FUNCTION_BLOCK L0_8070Service (* FAGOR 8070 CNC service FB *)
  (* Standard: 61499-2; Description: This FB is the entry point of the CNC service *)
  (* Version 0.0, 2014-09-01, EQUEROL, UJI *)
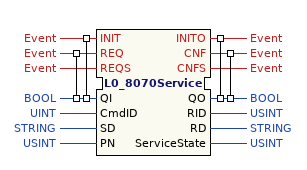
  EVENT_INPUT
    INIT WITH QI; (* Initialization Request *)
    REQ WITH QI; (* Normal Execution Request *)
    REQS; (* Request Service state *)
  END_EVENT
  EVENT_OUTPUT
    INITO WITH QO; (* Initialization Confirm *)
    CNF WITH QO; (* Execution Confirmation *)
    CNFS; (* Service State Confirmation *)
  END_EVENT
  VAR_INPUT
    QI : BOOL; (* Input event qualifier *)
    CmdID : UINT; (* Action to be executed ID *)
    SD : STRING; (* Action parameters *)
    PN : USINT; (* Number of parameters *)
  END_VAR
  VAR_OUTPUT
    QO : BOOL; (* Output event qualifier *)
    RID : USINT; (* Executed action ID *)
    RD : STRING; (* Service feedback data *)
    ServiceState : USINT; (* CNC Service state *)
  END_VAR
  FBS
    L0_State : L0_State;
    L0_SendBlk : L0_SendBlk;
    L0_CNCEncap : L0_CNCEncap;
    L0_IncomEx : L0_IncomEx;
    L0_StateHandler : L0_StateHandler;
    L0_CompletedEx : L0_CompletedEx;
    CM_Merge2E2USINT : CM_Merge2E2USINT;
    CM_Merge2E2USINT_0 : CM_Merge2E2USINT(E1In := 3, E2In := 4);
    CM_ChkService : CM_ChkService;
    CM_Merge2E2USINT_1 : CM_Merge2E2USINT;
    L0_ReqManager : L0_ReqManager;
    L0_InitService : L0_InitService;
  END_FBS
  EVENT_CONNECTIONS
    L0_SendBlk.IND TO L0_State.UPDT;
    L0_CNCEncap.CNF TO L0_SendBlk.REQ;
    L0_CNCEncap.INITO TO L0_SendBlk.INIT;
    L0_SendBlk.INITO TO L0_State.INIT;
    L0_StateHandler.OnInterrupted TO L0_IncomEx.Interrupted;
    L0_StateHandler.OnIntError TO L0_IncomEx.InterrupErr;
    L0_StateHandler.OnReady TO L0_CompletedEx.OnReady;
    L0_StateHandler.OnExecution TO L0_CompletedEx.OnExecuting;
    L0_StateHandler.OnNotReady TO L0_CompletedEx.OnNotReady;
    L0_CompletedEx.Success TO CM_Merge2E2USINT.E1;
    L0_IncomEx.CNF TO CM_Merge2E2USINT.E2;
    L0_State.UPDTO TO L0_StateHandler.REQ;
    CM_ChkService.BUSY TO CM_Merge2E2USINT_0.E2;
    CM_ChkService.DOWN TO CM_Merge2E2USINT_0.E1;
    CM_ChkService.UP TO L0_ReqManager.REQ;
    CM_ChkService.REQS TO L0_State.REQ;
    CM_Merge2E2USINT_0.EO TO CM_Merge2E2USINT_1.E2;
    L0_ReqManager.IND TO CM_Merge2E2USINT_1.E1;
    CM_Merge2E2USINT.EO TO L0_ReqManager.UPDT;
    CM_Merge2E2USINT_1.EO TO CNF;
    REQS TO L0_State.REQ;
    L0_State.CNF TO CNFS;
    L0_State.CNF TO CM_ChkService.RSP;
    REQ TO CM_ChkService.REQ;
    INIT TO L0_InitService.INIT;
    L0_InitService.INITOSer TO L0_ReqManager.INIT;
    L0_ReqManager.INITO TO L0_CNCEncap.INIT;
    L0_State.INITO TO L0_InitService.INITSer;
    L0_InitService.INITO TO INITO;
  END_CONNECTIONS
  DATA_CONNECTIONS
    L0_SendBlk.CNCState TO L0_State.StateIn;
    CmdID TO L0_CNCEncap.CmdID;
    SD TO L0_CNCEncap.SD;
    PN TO L0_CNCEncap.PN;
    L0_CNCEncap.sBlock TO L0_SendBlk.sBlock;
    L0_CNCEncap.QO TO L0_SendBlk.QI;
    L0_CompletedEx.RID TO CM_Merge2E2USINT.E1In;
    L0_IncomEx.RID TO CM_Merge2E2USINT.E2In;
    L0_State.StateOut TO L0_StateHandler.CNCState;
    CM_Merge2E2USINT_0.Out TO CM_Merge2E2USINT_1.E2In;
    L0_ReqManager.RIDOut TO CM_Merge2E2USINT_1.E1In;
    CM_Merge2E2USINT.Out TO L0_ReqManager.RIDIn;
    CM_Merge2E2USINT_1.Out TO RID;
    L0_State.ServiceState TO CM_ChkService.ServiceSate;
    L0_State.ServiceState TO ServiceState;
    L0_InitService.QO2 TO L0_ReqManager.QI;
    L0_ReqManager.QO TO L0_CNCEncap.QI;
    L0_InitService.QO1 TO QO;
    QI TO L0_InitService.QI1;
  END_CONNECTIONS
END_FUNCTION_BLOCK
